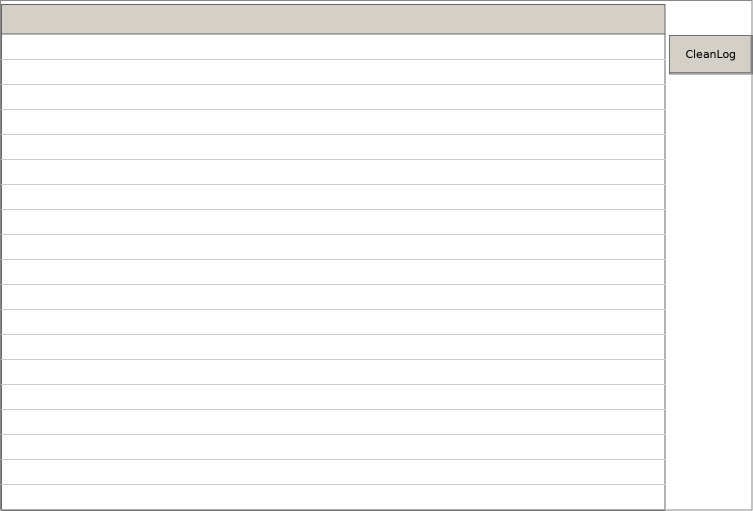
VISUALIZATION Visualization_LogEvent  // 753x511
    Button (669,35 84x39), "CleanLog"
        tap Alm_bHMIClearHistory
    Table (1,4 664x507), data array: AlarmHistoryArray
        p3854506369: AlarmHistoryArray[INDEX].EventMessage
        p1892666644: AlarmHistoryArray[INDEX].EventId
        p338671338: AlarmHistoryArray[INDEX].EventTime
END_VISUALIZATION

(* stored: Version 1.1.0.1, ProductVersion 3.1.4024.11
   Visu Visualization_LogEvent: Id {75d90e49-027d-4dc9-a955-0cd98a81d801} *)
